// TIA Portal V17 program export: 0 tag tables, 0 data types, 0 data blocks, 6 code blocks (in call order from the OBs), 0 instance data blocks

ORGANIZATION_BLOCK "OB1_CYCLE"   // OB1, LAD, ProgramCycle
TITLE = "Main Program Sweep (Cycle)"
{ S7_Optimized_Access := 'FALSE' }
VERSION : 0.1
// stored: AutoNumber false, IsIECCheckEnabled false, SetENOAutomatically false
   VAR_TEMP
      EV_CLASS : Byte;   // Bits 0-3 = 1:Coming event, Bits 4-7 = 1:Event class 1
      SCAN_1 : Byte;   // 1:Initial call of the OB, 3: Call 2-n of the OB
      PRIORITY : Byte;   // Priority of OB Execution
      OB_NUMBR : Byte;   // OB number
      RESERVED_1 : Byte;   // Reserved for system
      RESERVED_2 : Byte;   // Reserved for system
      PREV_CYCLE : Int;   // Previous program cycle time (milliseconds)
      MIN_CYCLE : Int;   // Minimum program cycle time (milliseconds)
      MAX_CYCLE : Int;   // Maximum program cycle time (milliseconds)
      DATE_TIME : Date_And_Time;   // Date and time OB started
      OB1_SCAN : Byte;   // 1 (Cold restart scan 1 of OB 1), 3 (Scan 2-n of OB 1)
      OB1_PRIORITY : Int;   // Priority of OB Execution
      OB1_MIN_CYCLE : DInt;   // Minimum cycle time of OB1 (milliseconds)
      OB1_MAX_CYCLE : DInt;   // Maximum cycle time of OB1 (milliseconds)
      PART_TYPE : Int;
      zero : Byte;
      status_sfc21 : Int;
      Error : Bool;
      status : Word;
   END_VAR
   VAR_TEMP   // added for the SCL form of the ladder/FBD networks
      _w1 : Bool;
   END_VAR
BEGIN

REGION Network 1: M ZERO - M ONE
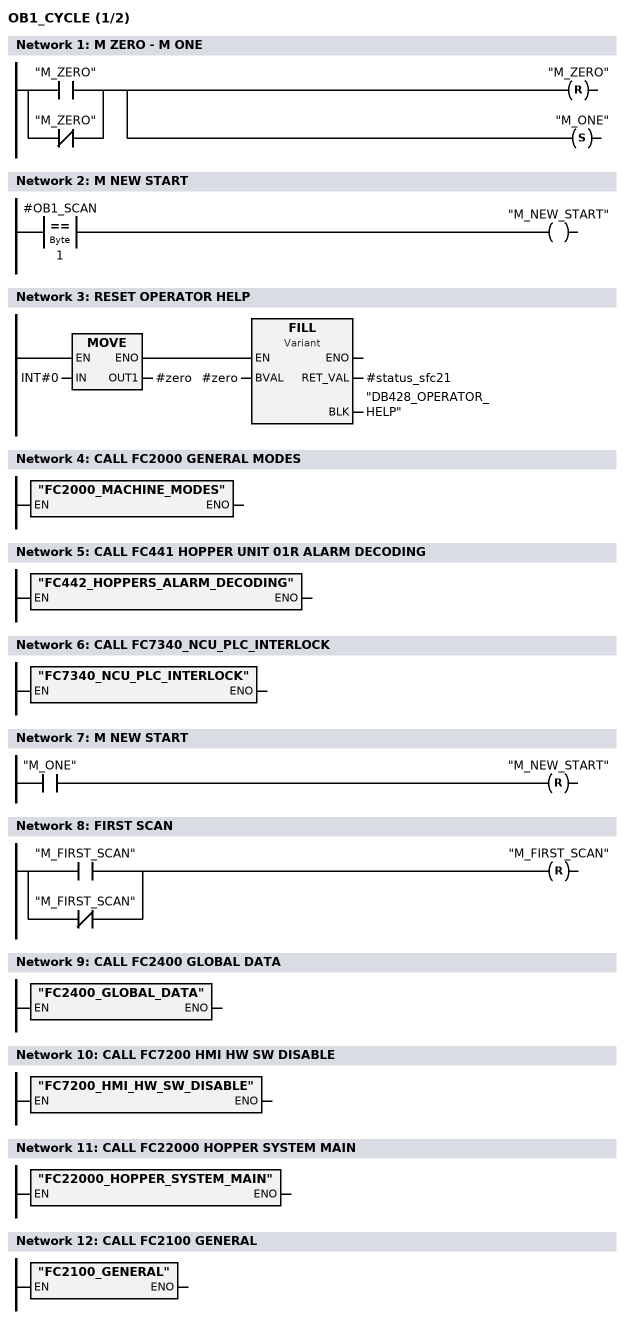
   RUNG wire#powerrail
      Contact( "M_ZERO" )
      wire#w1
      R_Coil( "M_ZERO" )
   END_RUNG
   RUNG wire#powerrail
      I_Contact( "M_ZERO" )
   END_RUNG wire#w1
   RUNG wire#w1
      S_Coil( "M_ONE" )
   END_RUNG
   // the same network as SCL:
   #_w1 := "M_ZERO" OR NOT "M_ZERO";
   IF #_w1 THEN
       "M_ZERO" := FALSE;
       "M_ONE" := TRUE;
   END_IF;
END_REGION

REGION Network 2: M NEW START
   RUNG wire#powerrail
      { S7_Templates := "SrcType := Byte" } EQ_Contact(in1 := #OB1_SCAN, in2 := 1)
      Coil( "M_NEW_START" )
   END_RUNG
   // the same network as SCL:
   "M_NEW_START" := #OB1_SCAN = 1;
END_REGION

REGION Network 3: RESET OPERATOR HELP
   RUNG wire#powerrail
      { S7_GenerateENO := "TRUE" } Move(in := INT#0, out1 => #zero)
      { S7_Templates := "ptr_type := Variant" } FILL(BVAL := #zero, RET_VAL => #status_sfc21, BLK => "DB428_OPERATOR_HELP")
   END_RUNG
   // the same network as SCL:
   // ENO of a box is taken as its EN; it also drops when the box reports an error
   #zero := INT#0;
   #status_sfc21 := FILL(BVAL := #zero, BLK => "DB428_OPERATOR_HELP");
END_REGION

REGION Network 4: CALL FC2000 GENERAL MODES
   RUNG wire#powerrail
      "FC2000_MACHINE_MODES"()
   END_RUNG
   // the same network as SCL:
   "FC2000_MACHINE_MODES"();
END_REGION

REGION Network 5: CALL FC441 HOPPER UNIT 01R ALARM DECODING
   RUNG wire#powerrail
      "FC442_HOPPERS_ALARM_DECODING"()
   END_RUNG
   // the same network as SCL:
   "FC442_HOPPERS_ALARM_DECODING"();
END_REGION

REGION Network 6: CALL FC7340_NCU_PLC_INTERLOCK
   RUNG wire#powerrail
      "FC7340_NCU_PLC_INTERLOCK"()
   END_RUNG
   // the same network as SCL:
   "FC7340_NCU_PLC_INTERLOCK"();
END_REGION

REGION Network 7: M NEW START
   RUNG wire#powerrail
      Contact( "M_ONE" )
      R_Coil( "M_NEW_START" )
   END_RUNG
   // the same network as SCL:
   IF "M_ONE" THEN "M_NEW_START" := FALSE; END_IF;
END_REGION

REGION Network 8: FIRST SCAN
   RUNG wire#powerrail
      Contact( "M_FIRST_SCAN" )
      wire#w1
      R_Coil( "M_FIRST_SCAN" )
   END_RUNG
   RUNG wire#powerrail
      I_Contact( "M_FIRST_SCAN" )
   END_RUNG wire#w1
   // the same network as SCL:
   IF "M_FIRST_SCAN" OR NOT "M_FIRST_SCAN" THEN "M_FIRST_SCAN" := FALSE; END_IF;
END_REGION

REGION Network 9: CALL FC2400 GLOBAL DATA
   RUNG wire#powerrail
      "FC2400_GLOBAL_DATA"()
   END_RUNG
   // the same network as SCL:
   "FC2400_GLOBAL_DATA"();
END_REGION

REGION Network 10: CALL FC7200 HMI HW SW DISABLE
   RUNG wire#powerrail
      "FC7200_HMI_HW_SW_DISABLE"()
   END_RUNG
   // the same network as SCL:
   "FC7200_HMI_HW_SW_DISABLE"();
END_REGION

REGION Network 11: CALL FC22000 HOPPER SYSTEM MAIN
   RUNG wire#powerrail
      "FC22000_HOPPER_SYSTEM_MAIN"()
   END_RUNG
   // the same network as SCL:
   "FC22000_HOPPER_SYSTEM_MAIN"();
END_REGION

REGION Network 12: CALL FC2100 GENERAL
   RUNG wire#powerrail
      "FC2100_GENERAL"()
   END_RUNG
   // the same network as SCL:
   "FC2100_GENERAL"();
END_REGION

REGION Network 13: CALL FC21000 POWDER FEEDER MAIN
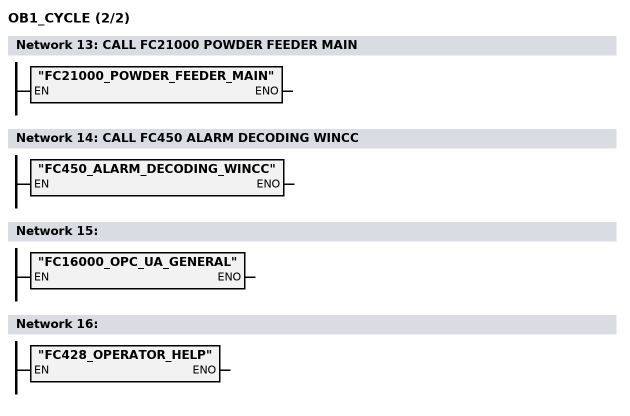
   RUNG wire#powerrail
      "FC21000_POWDER_FEEDER_MAIN"()
   END_RUNG
   // the same network as SCL:
   "FC21000_POWDER_FEEDER_MAIN"();
END_REGION

REGION Network 14: CALL FC450 ALARM DECODING WINCC
   RUNG wire#powerrail
      "FC450_ALARM_DECODING_WINCC"()
   END_RUNG
   // the same network as SCL:
   "FC450_ALARM_DECODING_WINCC"();
END_REGION

REGION Network 15
   RUNG wire#powerrail
      "FC16000_OPC_UA_GENERAL"()
   END_RUNG
   // the same network as SCL:
   "FC16000_OPC_UA_GENERAL"();
END_REGION

REGION Network 16
   RUNG wire#powerrail
      "FC428_OPERATOR_HELP"()
   END_RUNG
   // the same network as SCL:
   "FC428_OPERATOR_HELP"();
END_REGION
END_ORGANIZATION_BLOCK

ORGANIZATION_BLOCK "Cyclic interrupt"   // OB30, LAD, CyclicInterrupt
{ S7_Optimized_Access := 'TRUE' }
VERSION : 0.1
// stored: AutoNumber false, IsIECCheckEnabled false, SetENOAutomatically false
   VAR_INPUT
      Initial_Call : Bool;   // Initial call of this OB
      Event_Count : Int;   // Events discarded
   END_VAR
   VAR_TEMP
      LOOP_COUNT : Int;
   END_VAR
BEGIN

REGION Network 1: INITIALIZING OF ARRAY POINTERS FOR LOOP / Initializing of array pointers for loop
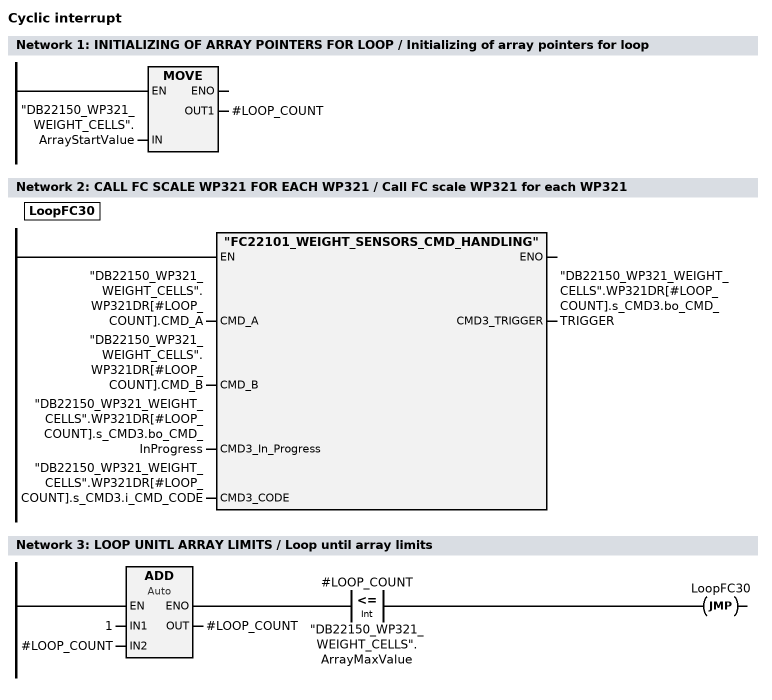
   RUNG wire#powerrail
      Move(in := "DB22150_WP321_WEIGHT_CELLS".ArrayStartValue, out1 => #LOOP_COUNT)
   END_RUNG
   // the same network as SCL:
   #LOOP_COUNT := "DB22150_WP321_WEIGHT_CELLS".ArrayStartValue;
END_REGION

REGION Network 2: CALL FC SCALE WP321 FOR EACH WP321 / Call FC scale WP321 for each WP321
   Label( LoopFC30 )
   RUNG wire#powerrail
      "FC22101_WEIGHT_SENSORS_CMD_HANDLING"(CMD_A := "DB22150_WP321_WEIGHT_CELLS".WP321DR[#LOOP_COUNT].CMD_A, CMD_B := "DB22150_WP321_WEIGHT_CELLS".WP321DR[#LOOP_COUNT].CMD_B, CMD3_In_Progress := "DB22150_WP321_WEIGHT_CELLS".WP321DR[#LOOP_COUNT].s_CMD3.bo_CMD_InProgress, CMD3_CODE := "DB22150_WP321_WEIGHT_CELLS".WP321DR[#LOOP_COUNT].s_CMD3.i_CMD_CODE, CMD3_TRIGGER => "DB22150_WP321_WEIGHT_CELLS".WP321DR[#LOOP_COUNT].s_CMD3.bo_CMD_TRIGGER)
   END_RUNG
   // the same network as SCL:
   LoopFC30:
   "FC22101_WEIGHT_SENSORS_CMD_HANDLING"(CMD_A := "DB22150_WP321_WEIGHT_CELLS".WP321DR[#LOOP_COUNT].CMD_A,
                           CMD_B := "DB22150_WP321_WEIGHT_CELLS".WP321DR[#LOOP_COUNT].CMD_B,
                           CMD3_In_Progress := "DB22150_WP321_WEIGHT_CELLS".WP321DR[#LOOP_COUNT].s_CMD3.bo_CMD_InProgress,
                           CMD3_CODE := "DB22150_WP321_WEIGHT_CELLS".WP321DR[#LOOP_COUNT].s_CMD3.i_CMD_CODE,
                           CMD3_TRIGGER => "DB22150_WP321_WEIGHT_CELLS".WP321DR[#LOOP_COUNT].s_CMD3.bo_CMD_TRIGGER);
END_REGION

REGION Network 3: LOOP UNITL ARRAY LIMITS / Loop until array limits
   RUNG wire#powerrail
      Add(in1 := 1, in2 := #LOOP_COUNT, out => #LOOP_COUNT)
      { S7_Templates := "SrcType := Int" } LE_Contact(in1 := #LOOP_COUNT, in2 := "DB22150_WP321_WEIGHT_CELLS".ArrayMaxValue)
      JumpCoil( LoopFC30 )
   END_RUNG
   // the same network as SCL:
   #LOOP_COUNT := 1 + #LOOP_COUNT;
   IF #LOOP_COUNT <= "DB22150_WP321_WEIGHT_CELLS".ArrayMaxValue THEN GOTO LoopFC30; END_IF;
END_REGION
END_ORGANIZATION_BLOCK

ORGANIZATION_BLOCK "OB100_RESTART"   // OB100, LAD, Startup
TITLE = "Complete Restart"
{ S7_Optimized_Access := 'FALSE' }
AUTHOR : ETXETAR
VERSION : 1.0
// stored: AutoNumber false, IsIECCheckEnabled false, SetENOAutomatically false
   VAR_TEMP
      OB100_EV_CLASS : Byte;
      OB100_STRTUP : Byte;
      OB100_PRIORITY : Byte;
      OB100_OB_NUMBR : Byte;
      OB100_RESERVED_1 : Byte;
      OB100_RESERVED_2 : Byte;
      OB100_STOP : Word;
      OB100_RESERVED_3 : Word;
      OB100_RESERVED_4 : Word;
      OB100_DATE_TIME : Date_And_Time;
      __PlcmigTempFillBits_20B0 : Array[0..7] of Bool;
   END_VAR
BEGIN

REGION Network 1: M_ONE / ESTABLISH "LOGIC 1" BIT
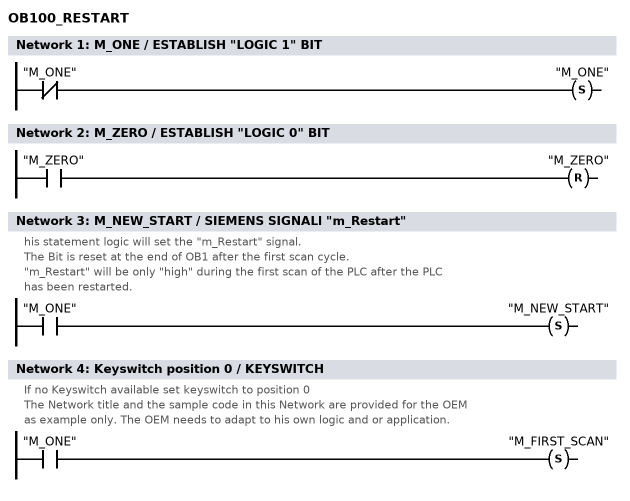
   RUNG wire#powerrail
      I_Contact( "M_ONE" )
      S_Coil( "M_ONE" )
   END_RUNG
   // the same network as SCL:
   IF NOT "M_ONE" THEN "M_ONE" := TRUE; END_IF;
END_REGION

REGION Network 2: M_ZERO / ESTABLISH "LOGIC 0" BIT
   RUNG wire#powerrail
      Contact( "M_ZERO" )
      R_Coil( "M_ZERO" )
   END_RUNG
   // the same network as SCL:
   IF "M_ZERO" THEN "M_ZERO" := FALSE; END_IF;
END_REGION

REGION Network 3: M_NEW_START / SIEMENS SIGNALl "m_Restart"
   // his statement logic will set the "m_Restart" signal.
   // The Bit is reset at the end of OB1 after the first scan cycle.
   // 
   // "m_Restart" will be only "high" during the first scan of the PLC after the PLC 
   // has been restarted.
   RUNG wire#powerrail
      Contact( "M_ONE" )
      S_Coil( "M_NEW_START" )
   END_RUNG
   // the same network as SCL:
   IF "M_ONE" THEN "M_NEW_START" := TRUE; END_IF;
END_REGION

REGION Network 4: Keyswitch position 0 / KEYSWITCH
   // If no Keyswitch available set keyswitch to position 0
   // 
   // The Network title and the sample code in this Network are provided for the OEM 
   // as example only. The OEM needs to adapt to his own logic and or application.
   RUNG wire#powerrail
      Contact( "M_ONE" )
      S_Coil( "M_FIRST_SCAN" )
   END_RUNG
   // the same network as SCL:
   IF "M_ONE" THEN "M_FIRST_SCAN" := TRUE; END_IF;
END_REGION
END_ORGANIZATION_BLOCK

ORGANIZATION_BLOCK "OB121_SYNCHRONF1"   // OB121, LAD, ProgrammingError
{ S7_Optimized_Access := 'FALSE' }
VERSION : 0.0
// stored: IsIECCheckEnabled false, SetENOAutomatically false
   VAR_TEMP
      TEMP0 : Byte;
      TEMP1 : Byte;
      TEMP2 : Byte;
      TEMP3 : Byte;
      TEMP4 : Byte;
      TEMP5 : Byte;
      TEMP6 : Word;
      TEMP7 : Word;
      TEMP8 : Word;
      TEMP9 : Date_And_Time;
   END_VAR
BEGIN
END_ORGANIZATION_BLOCK

ORGANIZATION_BLOCK "OB122_SYNCHRONF2"   // OB122, LAD, IOAccessError
{ S7_Optimized_Access := 'FALSE' }
VERSION : 0.0
// stored: IsIECCheckEnabled false, SetENOAutomatically false
   VAR_TEMP
      TEMP0 : Byte;
      TEMP1 : Byte;
      TEMP2 : Byte;
      TEMP3 : Byte;
      TEMP4 : Byte;
      TEMP5 : Byte;
      TEMP6 : Word;
      TEMP7 : Word;
      TEMP8 : Word;
      TEMP9 : Date_And_Time;
   END_VAR
BEGIN
END_ORGANIZATION_BLOCK

ORGANIZATION_BLOCK "OB40 Hardware interrupt"   // OB40, LAD, HardwareInterrupt
{ S7_Optimized_Access := 'TRUE' }
VERSION : 0.1
// stored: AutoNumber true, IsIECCheckEnabled false, SetENOAutomatically false
   VAR_INPUT
      LADDR : HW_IO;   // Hardware identifier
      USI : Word;   // User structure identifier
      IChannel : USInt;   // Interrupt channel number
      EventType : Byte;   // EventType
      PointAddr : DWord;
   END_VAR
   VAR_TEMP
      FLAG : Variant;
   END_VAR
BEGIN
END_ORGANIZATION_BLOCK
